PROGRAM PB_TestRunner
VAR
    TestRunner : T_TestRunner;
    Init : BOOL := TRUE;
END_VAR

IF TestRunner.ReloadTests OR Init THEN
    TestRunner.ClearTests();
    TestRunner.AddTestSuite(UnitTests.ExecutionTests);
    TestRunner.AddTestSuite(UnitTests.FunctionTests);
    TestRunner.AddTestSuite(UnitTests.StreamTests);
    TestRunner.AddTestSuite(UnitTests.NotificationTests);
    
    TestRunner.ReloadTests := Init := FALSE;
END_IF

TestRunner();

END_PROGRAM

(* stored: Version 1.1.0.1, ProductVersion 3.1.4024.9
   POU PB_TestRunner: Id {fcbfbb76-97bd-42a3-aa55-5d0eee0bed17}, SpecialFunc None *)
